FUNCTION_BLOCK items2Array (* Basic Function Block Type *)
  (* Standard: 61499-2 *)
  (* Version 0.0, 19/09/2015, kollger, nxtControl GmbH, Template *)
  PACKAGE Main;
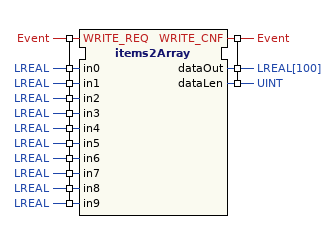
  EVENT_INPUT
    WRITE_REQ WITH in0, in1, in2, in3, in4, in5, in6, in7, in8, in9;
  END_EVENT
  EVENT_OUTPUT
    WRITE_CNF WITH dataOut, dataLen; (* Execution Confirmation *)
  END_EVENT
  VAR_INPUT
    in0 : LREAL; (* Input event qualifier *)
    in1 : LREAL;
    in2 : LREAL;
    in3 : LREAL;
    in4 : LREAL;
    in5 : LREAL;
    in6 : LREAL;
    in7 : LREAL;
    in8 : LREAL;
    in9 : LREAL;
  END_VAR
  VAR_OUTPUT
    dataOut : ARRAY [0..99] OF LREAL; (* Output event qualifier *)
    dataLen : UINT;
  END_VAR
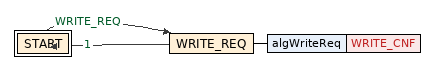
  EC_STATES
    START; (* Initial State *)
    WRITE_REQ : algWriteReq -> WRITE_CNF; (* Normal execution *)
  END_STATES
  EC_TRANSITIONS
    START TO WRITE_REQ := WRITE_REQ;
    WRITE_REQ TO START := 1;
  END_TRANSITIONS
  ALGORITHM algWriteReq IN ST: (* Normally executed algorithm *)
dataOut[0] := in0;
dataOut[1] := in1;
dataOut[2] := in2;
dataOut[3] := in3;
dataOut[4] := in4;
dataOut[5] := in5;
dataOut[6] := in6;
dataOut[7] := in7;
dataOut[8] := in8;
dataOut[9] := in9;

dataLen := 10;
  END_ALGORITHM
END_FUNCTION_BLOCK
